FUNCTION_BLOCK C_GenericDigital_2Channel IMPLEMENTS IFC_GENERIC_IO_INTERFACE
VAR_INPUT
END_VAR
VAR_OUTPUT
END_VAR
VAR
	Channel_Data AT %Q* : ARRAY[1..2] OF BOOL;
END_VAR

METHOD IO_Read : ph_lv0.RETURN_CODE
VAR_INPUT
	CHANNEL	: INT;
	DATA	: POINTER TO LREAL;
END_VAR
END_METHOD

{warning 'add property implementation'}
PROPERTY IO_TYPE : INT
GET
END_GET
SET
END_SET
END_PROPERTY

{warning 'add method implementation'}
METHOD IO_Write : ph_lv0.RETURN_CODE
VAR_INPUT
	CHANNEL	: INT;
	DATA	: LREAL;
END_VAR
END_METHOD

END_FUNCTION_BLOCK

(* stored: Version 1.1.0.1, ProductVersion 3.1.4019.2
   POU C_GenericDigital_2Channel: Id {d84c7027-fcca-4afa-8053-19d979d3531b}, SpecialFunc None
   Method IO_Read: Id {adbcf430-ee4a-4ada-858b-f3f90cd33617}
   Property IO_TYPE: Id {4089dc1e-1971-47de-96e1-a1ac2a1a61b7}
   Get Get: Id {974d94e8-0491-4a76-b01e-ee2cee225380}
   Set Set: Id {ba07c148-1785-4a3f-8b94-1a3023c65639}
   Method IO_Write: Id {a9af7171-8e03-4ddc-a682-38807e7524b6} *)
